FUNCTION_BLOCK PUMP_POWER

VAR_INPUT
	PUMP_STATUS	:INT;
	EMS_OK			:BOOL;
END_VAR

VAR_OUTPUT
	POWER			:BOOL;
	POWER_LED	:BOOL;
END_VAR

VAR
END_VAR

IF PUMP_STATUS=1 AND EMS_OK THEN

POWER:=TRUE;
POWER_LED:=TRUE;

ELSE

POWER:=FALSE;
POWER_LED:=FALSE;

END_IF;

END_FUNCTION_BLOCK

(* stored: Version 1.1.0.1, ProductVersion 3.1.0.26
   POU PUMP_POWER: Id {7736fa49-7bbe-42c0-8b4b-dd20ce02697d} *)
